INTERFACE ICheckEofActionCallback EXTENDS __SYSTEM.IQueryInterface

METHOD OnActionComplete
VAR_INPUT
	actionId : UINT;
	isEOF : BOOL;
END_VAR
END_METHOD

END_INTERFACE

(* stored: Version 1.1.0.1
   Itf ICheckEofActionCallback: Id {32d3cb20-19ce-44b1-84c3-13e423d7a75a}
   Method OnActionComplete: Id {952f33b2-bcad-4060-8eaa-db303a3407e9} *)
